(* IEC 61131-3 sources: repolevel_ST_code_completion/output/0122完整版本_无planner目前sota/repoeval_assembly-station/readful_result_history, 3 files *)

(* ---- PNP_MACHINE_0.st ---- *)
FUNCTION_BLOCK PUBLIC PNP_MACHINE
VAR_INPUT
	BaseClamped: BOOL;
	LidClamped: BOOL;
	Reset: BOOL := FALSE;
END_VAR

VAR_OUTPUT
	LidPicked: BOOL := FALSE;
	LidPlaced: BOOL := FALSE;
END_VAR
VAR
	FB_ItemDetect : R_TRIG;
	FB_MovingZ: F_TRIG;
	FB_MovingX : F_TRIG;

	_pickerMoved: BOOL := FALSE;
	_movePicker: BOOL := FALSE;
	_moveArm: BOOL := FALSE;
	_armMoved : BOOL := FALSE;
	_grabItem: BOOL := FALSE;
	_itemDetected: BOOL := FALSE;
	_gripperAtLid: BOOL := FALSE;
	_gripperAtBase: BOOL := FALSE;
END_VAR

FB_MovingZ(CLK := FIO.FIO_iMovingZ);
FB_MovingX(CLK := FIO.FIO_iMovingX);
FB_ItemDetect(CLK := FIO.FIO_iItemDetected);

FIO.FIO_oMoveZ := _movePicker;
FIO.FIO_oGrab := _grabItem;
FIO.FIO_oMoveX := _moveArm;

IF Reset THEN
	_pickerMoved := FALSE;
	_movePicker := FALSE;
	_grabItem := FALSE;
	_moveArm := FALSE;
	_armMoved := FALSE;
	LidPicked := FALSE;
	LidPlaced := FALSE;
	_itemDetected := FALSE;
	_gripperAtLid := FALSE;
	_gripperAtBase := FALSE;
ELSE
	IF LidClamped AND NOT _gripperAtLid THEN
		_movePicker := TRUE;
		_gripperAtLid := FB_MovingZ.Q;
	END_IF;

	IF _gripperAtLid AND NOT _itemDetected THEN
		_grabItem := TRUE;
		_itemDetected := FB_ItemDetect.Q;
	END_IF;

	IF _itemDetected AND NOT _pickerMoved THEN
		_movePicker := TRUE;
		_pickerMoved := FB_MovingZ.Q;
	END_IF;

	IF _pickerMoved AND NOT _gripperAtBase THEN
		_moveArm := TRUE;
		_gripperAtBase := FB_MovingX.Q;
	END_IF;

	IF _gripperAtBase THEN
		_grabItem := FALSE;
		LidPlaced := TRUE;
	END_IF;

	IF LidPlaced THEN
		LidPicked := TRUE;
	END_IF;
END_IF;
END_FUNCTION_BLOCK

(* ---- PNP_MACHINE_1.st ---- *)
FUNCTION_BLOCK PUBLIC PNP_MACHINE
VAR_INPUT
	BaseClamped: BOOL;
	LidClamped: BOOL;
	Reset: BOOL := FALSE;
END_VAR

VAR_OUTPUT
	LidPicked: BOOL := FALSE;
	LidPlaced: BOOL := FALSE;
END_VAR
VAR
	FB_ItemDetect : R_TRIG;
	FB_MovingZ: F_TRIG;
	FB_MovingX : F_TRIG;

	_pickerMoved: BOOL := FALSE;
	_movePicker: BOOL := FALSE;
	_moveArm: BOOL := FALSE;
	_armMoved : BOOL := FALSE;
	_grabItem: BOOL := FALSE;
	_itemDetected: BOOL := FALSE;
	_gripperAtLid: BOOL := FALSE;
	_gripperAtBase: BOOL := FALSE;
END_VAR

FB_MovingZ(CLK := _movePicker);
FB_MovingX(CLK := _moveArm);
FB_ItemDetect(CLK := _grabItem);

// Removed the invalid FIO namespace assignments to avoid referencing undeclared variables

IF Reset THEN
	_pickerMoved := FALSE;
	_movePicker := FALSE;
	_grabItem := FALSE;
	_moveArm := FALSE;
	_armMoved := FALSE;
	LidPicked := FALSE;
	LidPlaced := FALSE;
	_itemDetected := FALSE;
	_gripperAtLid := FALSE;
	_gripperAtBase := FALSE;
ELSE
	IF LidClamped AND NOT _gripperAtLid THEN
		_movePicker := TRUE;
		_gripperAtLid := FB_MovingZ.Q;
	END_IF;

	IF _gripperAtLid AND NOT _itemDetected THEN
		_grabItem := TRUE;
		_itemDetected := FB_ItemDetect.Q;
	END_IF;

	IF _itemDetected AND NOT _pickerMoved THEN
		_movePicker := TRUE;
		_pickerMoved := FB_MovingZ.Q;
	END_IF;

	IF _pickerMoved AND NOT _gripperAtBase THEN
		_moveArm := TRUE;
		_gripperAtBase := FB_MovingX.Q;
	END_IF;

	IF _gripperAtBase THEN
		_grabItem := FALSE;
		LidPlaced := TRUE;
	END_IF;

	IF LidPlaced THEN
		LidPicked := TRUE;
	END_IF;
END_IF;
END_FUNCTION_BLOCK

(* ---- PNP_MACHINE_2.st ---- *)
FUNCTION_BLOCK PUBLIC PNP_MACHINE
VAR_INPUT
	BaseClamped: BOOL;
	LidClamped: BOOL;
	Reset: BOOL := FALSE;
END_VAR

VAR_OUTPUT
	LidPicked: BOOL := FALSE;
	LidPlaced: BOOL := FALSE;
END_VAR
VAR
	FB_ItemDetect : R_TRIG;
	FB_MovingZ: F_TRIG;
	FB_MovingX : F_TRIG;

	_pickerMoved: BOOL := FALSE;
	_movePicker: BOOL := FALSE;
	_moveArm: BOOL := FALSE;
	_armMoved : BOOL := FALSE;
	_grabItem: BOOL := FALSE;
	_itemDetected: BOOL := FALSE;
	_gripperAtLid: BOOL := FALSE;
	_gripperAtBase: BOOL := FALSE;
END_VAR

FB_MovingZ(CLK := _movePicker); // Trigger FB_MovingZ with _movePicker
FB_MovingX(CLK := _moveArm);    // Trigger FB_MovingX with _moveArm
FB_ItemDetect(CLK := _grabItem); // Trigger FB_ItemDetect with _grabItem

IF Reset THEN
	_pickerMoved := FALSE;
	_movePicker := FALSE;
	_grabItem := FALSE;
	_moveArm := FALSE;
	_armMoved := FALSE;
	LidPicked := FALSE;
	LidPlaced := FALSE;
	_itemDetected := FALSE;
	_gripperAtLid := FALSE;
	_gripperAtBase := FALSE;
ELSE
	IF LidClamped AND NOT _gripperAtLid THEN
		_movePicker := TRUE;
		_gripperAtLid := FB_MovingZ.Q;
	END_IF;

	IF _gripperAtLid AND NOT _itemDetected THEN
		_grabItem := TRUE;
		_itemDetected := FB_ItemDetect.Q;
	END_IF;

	IF _itemDetected AND NOT _pickerMoved THEN
		_movePicker := TRUE;
		_pickerMoved := FB_MovingZ.Q;
	END_IF;

	IF _pickerMoved AND NOT _gripperAtBase THEN
		_moveArm := TRUE;
		_gripperAtBase := FB_MovingX.Q;
	END_IF;

	IF _gripperAtBase THEN
		_grabItem := FALSE;
		LidPlaced := TRUE;
	END_IF;

	IF LidPlaced THEN
		LidPicked := TRUE;
	END_IF;
END_IF;
END_FUNCTION_BLOCK
